// Mitsubishi GX Works2 project: 자기유지   PLC: Q02/Q02H

PROGRAM MAIN
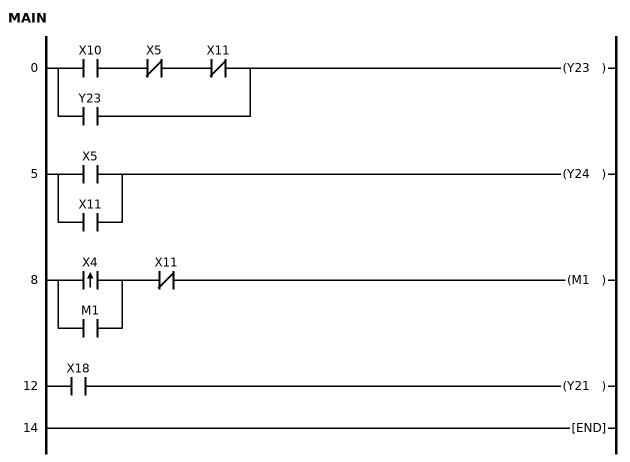
0     LD      X10
      ANI     X5
      ANI     X11
      OR      Y23
      OUT     Y23
5     LD      X5
      OR      X11
      OUT     Y24
8     LDP     X4
      OR      M1
      ANI     X11
      OUT     M1
12    LD      X18
      OUT     Y21
14    END
END_PROGRAM
